RoboDK station: DHEXP.rdk

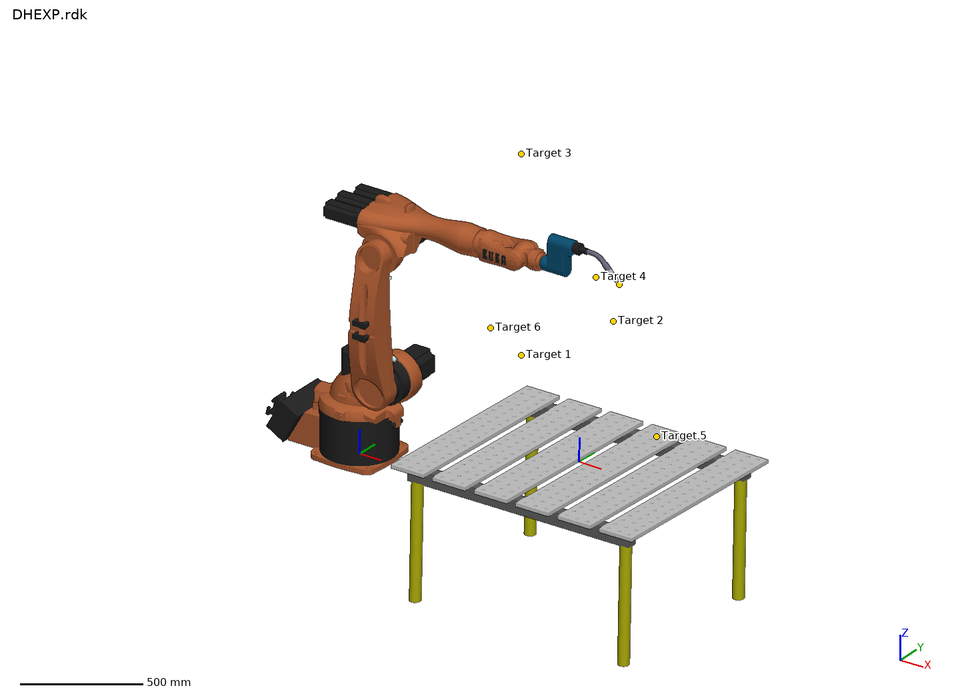
[picture v0: the station drawn from its stored meshes, robots at their saved joint values, targets as dots, program paths as lines]
Station DHEXP (saved by RoboDK 5.7.1). Poses are relative to the parent item; angles as X-Y-Z fixed-axis rotations.
  - frame KUKA KR 5 arc Base at (0, 0, 0) mm
    - robot KUKA KR 5 arc: 6 axes, payload 5 kg, reach 1411 mm, repeatability 0.04 mm, weight 127 kg
        modified DH rows (alpha deg, a mm, theta deg, d mm): 0, 0, 0, 400; -90, 180, 0, 0; 0, 600, -90, 0; -90, 120, 0, 620; 90, 0, 0, 0; -90, 0, 180, 115
        joint limits [-155, -180, -15, -350, -130, -350] to [155, 65, 158, 350, 130, 350]; home [0, -90, 90, 0, 0, 0]; saved at [0, -90, 90, 0, 0, 0]
      - tool Weld gun, TCP at (-4, 0, 371.3) mm, rotated rx 0 ry 45 rz 0 deg, size 299.9 x 60 x 318.3 mm
    - target Target 1 (Cartesian target) at (799.65, 4.79, 666.2) mm, rotated rx 180 ry 30 rz -180 deg; joints [-0.834, -143.424, 151.595, 186.745, -6.878, -186.913] of KUKA KR 5 arc
    - target Target 2 (Cartesian target) at (1253.88, 4.79, 947.15) mm, rotated rx 179.57 ry 47.27 rz 171.79 deg; joints [-5.297, -92.957, 110.758, -34.261, -23.918, -327.851] of KUKA KR 5 arc
    - target Target 3 (Cartesian target) at (800.31, 4.79, 1573.37) mm, rotated rx 13.1 ry 13.33 rz 171.98 deg; joints [3.807, -113.521, 104.079, -170.637, 48.009, 6.626] of KUKA KR 5 arc
    - target Target 4 (Cartesian target) at (1169.42, 4.79, 1119.76) mm, rotated rx 179.57 ry 47.27 rz 171.79 deg; joints [-5.942, -100.604, 101.825, -255.868, 14.28, -104.297] of KUKA KR 5 arc
    - target Target 5 (Cartesian target) at (1469.47, 4.79, 486.69) mm, rotated rx 179.57 ry 47.27 rz 171.79 deg; joints [-4.146, -54.825, 108.322, -194.462, 56.668, -171.741] of KUKA KR 5 arc
    - target Target 6 (Cartesian target) at (1087.88, -622.5, 1119.76) mm, rotated rx 179.57 ry 47.27 rz 171.79 deg; joints [42.483, -88.215, 90.351, -277.058, -34.846, -83.276] of KUKA KR 5 arc
    - target Home (Cartesian target) at (1286.3, 0, 1124) mm, rotated rx -180 ry 45 rz -180 deg; joints [0, -90, 90, 0, 0, 0] of KUKA KR 5 arc
  - frame Frame 2 at (1183.5, -134.94, 347.41) mm, rotated rx -1.74 ry 0 rz 0 deg
    - object Object Table at (0, 0, 0) mm, size 1193.8 x 965.2 x 609.6 mm, geometry from Object Table.wrl
